// Block: PPrgArchive9

DATA_BLOCK PPrgArchive9
VERSION : 0.1
   NON_RETAIN
   VAR
      PRG : Array[801..900] of PPrg_Data;
   END_VAR

BEGIN
   // No initialization required
END_DATA_BLOCK
